FUNCTION_BLOCK OR (* Basic Function Block Type *)
  (* Standard: 61499-2 *)
  (* Version 0.2, 2003-12-04, JHC, Rockwell Automation, Renamed for better indexing. *)
  (* Version 0.1, 2002-11-05, JHC, Rockwell Automation, Corrected missing ST element in Algorithm REQ. *)
  (* Version 0.0, 2000-05-30, JHC, Rockwell Automation *)
  (* Compiler header: package fb.rt.pnp; *)
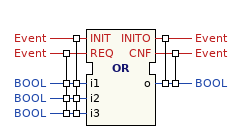
  EVENT_INPUT
    INIT WITH i1, i3, i2; (* Initialization Request *)
    REQ WITH i1, i2, i3; (* Normal Execution Request *)
  END_EVENT
  EVENT_OUTPUT
    INITO WITH o; (* Initialization Confirm *)
    CNF WITH o; (* Execution Confirmation *)
  END_EVENT
  VAR_INPUT
    i1 : BOOL; (* Input event qualifier *)
    i2 : BOOL;
    i3 : BOOL;
  END_VAR
  VAR_OUTPUT
    o : BOOL; (* Output event qualifier *)
  END_VAR
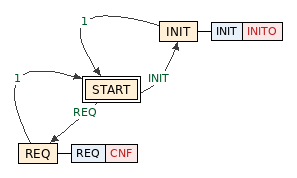
  EC_STATES
    START; (* Initial State *)
    INIT : INIT -> INITO; (* Initialization *)
    REQ : REQ -> CNF; (* Normal execution *)
  END_STATES
  EC_TRANSITIONS
    START TO INIT := INIT;
    INIT TO START := 1;
    START TO REQ := REQ;
    REQ TO START := 1;
  END_TRANSITIONS
  ALGORITHM INIT IN Java: (* Initialization algorithm *)
o.value=i1.value|i2.value|i3.value;
  END_ALGORITHM
  ALGORITHM REQ IN Java: (* Normally executed algorithm *)
o.value=i1.value|i2.value|i3.value;
  END_ALGORITHM
END_FUNCTION_BLOCK
